Staubli VAL3: start.pgx

program start()
begin
  call initCmdBuf()
  call FC_InitData()
  waitEndMove()
  taskCreate "tcprec",100,TcpStrRec:SockRec(datar,ststu)
  call InitSocket()

  taskCreate "CmdManage",100,CmdManage()
  taskCreate "HMI",99,HMI()
  taskCreate "CmdDeal",99,CmdDealTest()
  taskCreate "CmdTxtReading",85,CmdTxtReading()
end
